ADAPTER ABatteryModel
  (* Standard: 61499-1 *)
  (* Version 0.0, 2008-04-22, GE, 4DIAC-Consortium *)
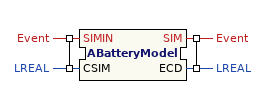
  EVENT_INPUT
    SIMIN WITH CSIM; (* Battery Simulation Arrival *)
  END_EVENT
  EVENT_OUTPUT
    SIM WITH ECD, ECD; (* Battery Simulation Request *)
  END_EVENT
  VAR_INPUT
    CSIM : LREAL; (* Battery capacity after simulation in kWh *)
  END_VAR
  VAR_OUTPUT
    ECD : LREAL; (* Charging (positive)/discharging (negative) energy for battery simulation in kWh *)
  END_VAR
  SERVICE SOCKET/PLUG
    SEQUENCE request_confirm
      SOCKET.REQ(REQD) -> PLUG.REQ(REQD);
      PLUG.CNF(CNFD) -> SOCKET.CNF(CNFD);
    END_SEQUENCE
    SEQUENCE indication_response
      PLUG.IND(INDD) -> SOCKET.IND(INDD);
      SOCKET.RSP(RSPD) -> PLUG.RSP(RSPD);
    END_SEQUENCE
  END_SERVICE
END_ADAPTER
